FUNCTION_BLOCK MovementController (* Basic Function Block Type *)
  (* Standard: 61499-2 *)
  (* Version 0.0, 9/23/2026, macie, Schneider Electric, Template *)
  PACKAGE Main;
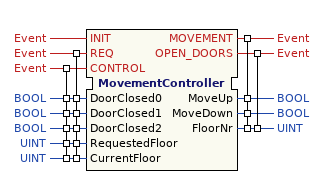
  EVENT_INPUT
    INIT; (* Initialization Request *)
    REQ WITH DoorClosed0, DoorClosed1, DoorClosed2, RequestedFloor, CurrentFloor; (* Normal Execution Request *)
    CONTROL WITH DoorClosed0, DoorClosed1, DoorClosed2, RequestedFloor, CurrentFloor;
  END_EVENT
  EVENT_OUTPUT
    MOVEMENT WITH MoveUp, MoveDown, FloorNr; (* Execution Confirmation *)
    OPEN_DOORS WITH FloorNr;
  END_EVENT
  VAR_INPUT
    DoorClosed0 : BOOL; (* Input event qualifier *)
    DoorClosed1 : BOOL;
    DoorClosed2 : BOOL;
    RequestedFloor : UINT;
    CurrentFloor : UINT;
  END_VAR
  VAR_OUTPUT
    MoveUp : BOOL := FALSE; (* Output event qualifier *)
    MoveDown : BOOL := FALSE;
    FloorNr : UINT := 2;
  END_VAR
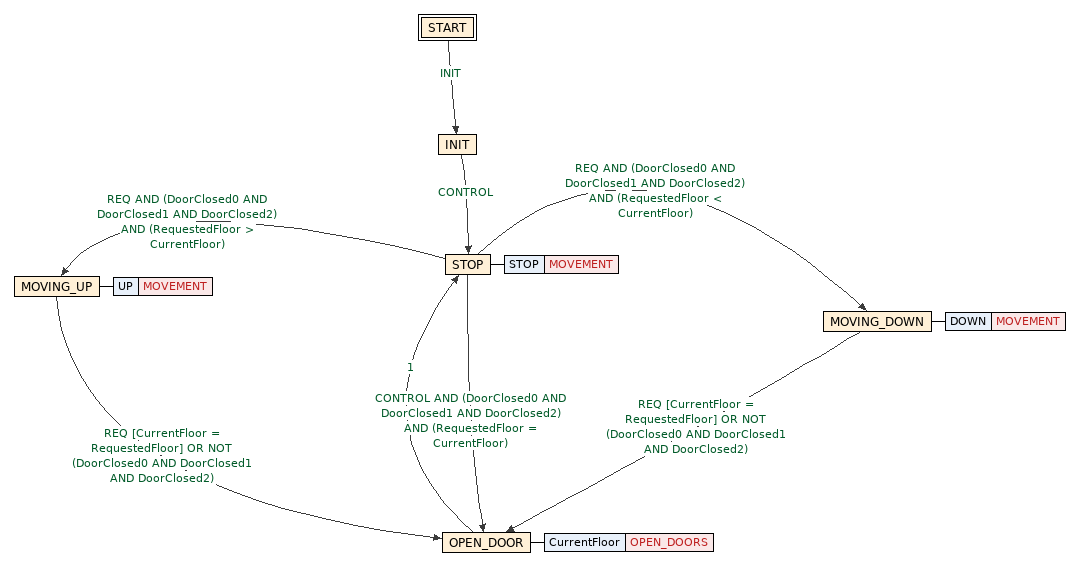
  EC_STATES
    START; (* Initial State *)
    STOP : STOP -> MOVEMENT;
    MOVING_UP : UP -> MOVEMENT;
    MOVING_DOWN : DOWN -> MOVEMENT;
    INIT;
    OPEN_DOOR : CurrentFloor -> OPEN_DOORS;
  END_STATES
  EC_TRANSITIONS
    STOP TO MOVING_DOWN := REQ AND (DoorClosed0 AND DoorClosed1 AND DoorClosed2) AND (RequestedFloor < CurrentFloor);
    MOVING_DOWN TO OPEN_DOOR := REQ [CurrentFloor = RequestedFloor] OR NOT (DoorClosed0 AND DoorClosed1 AND DoorClosed2);
    STOP TO MOVING_UP := REQ AND (DoorClosed0 AND DoorClosed1 AND DoorClosed2) AND (RequestedFloor > CurrentFloor);
    MOVING_UP TO OPEN_DOOR := REQ [CurrentFloor = RequestedFloor] OR NOT (DoorClosed0 AND DoorClosed1 AND DoorClosed2);
    START TO INIT := INIT;
    INIT TO STOP := CONTROL;
    STOP TO OPEN_DOOR := CONTROL AND (DoorClosed0 AND DoorClosed1 AND DoorClosed2) AND (RequestedFloor = CurrentFloor);
    OPEN_DOOR TO STOP := 1;
  END_TRANSITIONS
  ALGORITHM UP IN ST: (* Initialization algorithm *)
;
MoveUp := TRUE;
  END_ALGORITHM
  ALGORITHM DOWN IN ST: (* Normally executed algorithm *)
;
MoveDown := TRUE;
  END_ALGORITHM
  ALGORITHM STOP IN ST:
;
MoveDown := FALSE;
MoveUp := FALSE;
  END_ALGORITHM
  ALGORITHM CurrentFloor IN ST:
;
MoveDown := FALSE;
MoveUp := FALSE;
FloorNr := CurrentFloor;
  END_ALGORITHM
END_FUNCTION_BLOCK
